TYPE T_Long_String : STRING(255); END_TYPE

(* stored: Version 1.1.0.1, ProductVersion 3.1.4024.4
   DUT T_Long_String: Id {d57fe306-93a2-4aa3-9c36-026c7f90ffdc} *)
